FUNCTION_BLOCK FB_SR (* set dominant *)
  (* Standard: 61131-3; Classification: bistable function block; Description: Copyright (c) 2011 TU Wien ACIN This program and the accompanying materials are made available under the terms of the Eclipse Public License 2.0 which is available at https://www.eclipse.org/legal/epl-2.0/ SPDX-License-Identifier: EPL-2.0 *)
  (* Version 1.0, 2011-06-21, Monika Wenger, TU Wien ACIN *)
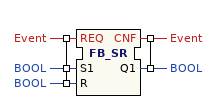
  EVENT_INPUT
    REQ WITH S1, R; (* Service Request *)
  END_EVENT
  EVENT_OUTPUT
    CNF WITH Q1; (* Confirmation of Requested Service *)
  END_EVENT
  VAR_INPUT
    S1 : BOOL; (* Set *)
    R : BOOL; (* Reset *)
  END_VAR
  VAR_OUTPUT
    Q1 : BOOL; (* Output *)
  END_VAR
  (* Service APPLICATION/RESOURCE: Bistable Function Block (set dominant) *)
END_FUNCTION_BLOCK
